{attribute 'qualified_only'}
{attribute 'strict'}
TYPE E_STATES :
(
	eState1 := 0,
	eState2
);
END_TYPE

(* stored: Version 1.1.0.1, ProductVersion 3.1.4024.3
   DUT E_STATES: Id {5c36365a-1b2a-4f7b-ba30-f0e6ea97731e} *)
